// TIA Portal V20 export
VAR_GLOBAL   // PLC tag table "Cognex"
   ASTriggerReady AT %I690.0 : Bool;   // Acquisition status
   ASTriggerAck AT %I690.1 : Bool;   // Acquisition status
   ASAcquiring AT %I690.2 : Bool;   // Acquisition status
   ASMissedTrig AT %I690.3 : Bool;   // Acquisition status
   ASOfflineResBit1 AT %I690.4 : Bool;   // Acquisition status
   ASOfflineResBit2 AT %I690.5 : Bool;   // Acquisition status
   ASOfflineResBit3 AT %I690.6 : Bool;   // Acquisition status
   ASOnline AT %I690.7 : Bool;   // Acquisition status
   ASAcquiNum AT %IW691 : Word;   // Acquisition status
   ISInspecting AT %I693.0 : Bool;   // Inspection status
   ISToggleInspectDone AT %I693.1 : Bool;   // Inspection status
   ISBufferOverrun AT %I693.2 : Bool;   // Inspection status
   ISResultsValid AT %I693.3 : Bool;   // Inspection status
   ISJobLoading AT %I693.4 : Bool;   // Inspection status
   ISJobLoadComplete AT %I693.5 : Bool;   // Inspection status
   ISJobLoadFailed AT %I693.6 : Bool;   // Inspection status
   ISSetUserDataACk AT %I693.7 : Bool;   // Inspection status
   ISJobPass AT %I694.0 : Bool;   // Inspection status
   SEC0Ack AT %I699.0 : Bool;   // Soft event control
   SEC1Ack AT %I699.1 : Bool;   // Soft event control
   SEC2Ack AT %I699.2 : Bool;   // Soft event control
   SEC3Ack AT %I699.3 : Bool;   // Soft event control
   SEC4Ack AT %I699.4 : Bool;   // Soft event control
   SEC5Ack AT %I699.5 : Bool;   // Soft event control
   SEC6Ack AT %I699.6 : Bool;   // Soft event control
   SEC7Ack AT %I699.7 : Bool;   // Soft event control
   JCJobID AT %IW697 : Word;   // Job control
   IRInspectionID AT %IW600 : Word;   // Inspection result
   IRInspectResultCode AT %IW602 : Word;   // Inspection result
   IRActHoleNrResult AT %IB606 : Byte;   // Inspection result
   ResultDataFromCognex0 AT %ID604 : DWord;
   ResultDataFromCognex1 AT %ID608 : DWord;
   ResultDataFromCognex2 AT %ID612 : DWord;
   ResultDataFromCognex3 AT %ID616 : DWord;
   ACTriggerEnable AT %Q690.0 : Bool;   // Acquisition control
   ACTrigger AT %Q690.1 : Bool;   // Acquisition control
   ACClearAcquirCompl AT %Q690.2 : Bool;   // Acquisition control
   ACSetOffline AT %Q690.7 : Bool;   // Acquisition control
   ICBufferResultsEn AT %Q691.0 : Bool;   // Inspection control
   ICInspectResultsAck AT %Q691.1 : Bool;   // Inspection control
   ICSetUserData AT %Q691.2 : Bool;   // Inspection control
   ICExecuteCmd AT %Q691.3 : Bool;   // Inspection control
   CCSetJobID AT %QW697 : Word;   // Command control
   SEC0 AT %Q699.0 : Bool;   // Soft event control
   SEC1 AT %Q699.1 : Bool;   // Soft event control
   SEC2 AT %Q699.2 : Bool;   // Soft event control
   SEC3 AT %Q699.3 : Bool;   // Soft event control
   SEC4 AT %Q699.4 : Bool;   // Soft event control
   SEC5 AT %Q699.5 : Bool;   // Soft event control
   SEC6 AT %Q699.6 : Bool;   // Soft event control
   SEC7 AT %Q699.7 : Bool;   // Soft event control
   UserDataToCognex0 AT %QD600 : DWord;
   UserDataToCognex1 AT %QD604 : DWord;
   UserDataToCognex2 AT %QD608 : DWord;
   UserDataToCognex3 AT %QD612 : DWord;
   UserDataToCognex4 AT %QD616 : DWord;
   UserDataToCognex5 AT %QD620 : DWord;
   UserDataToCognex6 AT %QD624 : DWord;
   UserDataToCognex7 AT %QD628 : DWord;
END_VAR
